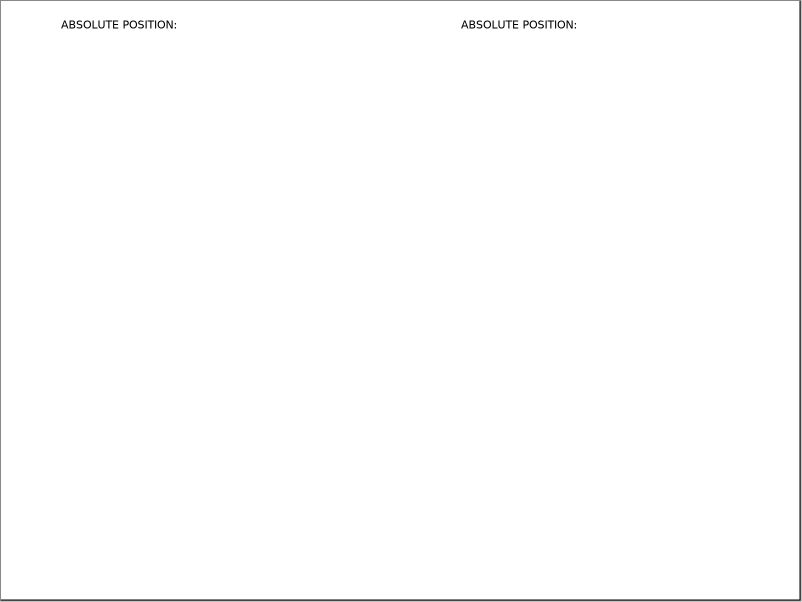
VISUALIZATION F37_Position_Profile  // 802x602
    Rectangle (0,0 800x600)
    Label (10,10 170x30), "ABSOLUTE POSITION:"
    Label (410,10 170x30), "ABSOLUTE POSITION:"
END_VISUALIZATION

(* stored: Version 1.1.0.1, ProductVersion 3.1.4022.7
   Visu F37_Position_Profile: Id {51904880-acd0-47a3-9407-5956e5b31a7e} *)
